// Disclaimer
// 
// This publication contains statements about the suitability of our products for certain areas of application. These statements are based on typical features of our products. The examples shown in this publication are for demonstration purposes only. 
// The information provided herein should not be regarded as specific operation characteristics. It is incumbent on the customer to check and decide whether a product is suitable for use in a particular application. 
// We do not give any warranty that the source code which is made available with this publication is complete or accurate. 
//
// THE SAMPLE CODE CONTAINED IN THIS PUBLICATION IS PROVIDED “AS IS” WITHOUT WARRANTY OF ANY KIND, EITHER EXPRESSED, IMPLIED OR STATUTORY, INCLUDING WITHOUT LIMITATION, ANY WARRANTY WITH RESPECT TO NON-INFRINGEMENT, FREEDOM FROM PROPRIETARY RIGHTS OF THIRD PARTIES OR FITNESS FOR ANY PARTICULAR PURPOSE. 
// This publication may be changed from time to time without prior notice. No liability is assumed for errors and/or omissions. Our products are described in detail in our data sheets and documentations. Product-specific warnings and cautions must be observed. 
// For the latest version of our data sheets and documentations visit our website (www.beckhoff.de). 
//
// © Beckhoff Automation GmbH & Co. KG, 2022
// The reproduction, distribution and utilization of this document as well as the communication of its contents to others without express authorization is prohibited. Offenders will be held liable for the payment of damages. All rights reserved in the event of the grant of a patent, utility model or design.
PROGRAM MAIN
VAR_INPUT
	bExecuteComplete			: BOOL;									//Command Execute Complete, not defined
END_VAR
VAR
	UserModeCofig				: PML_UnitModeConfig;					//User can configure his own Mode
	
	fbMachine					: FB_Machine;							//Instance of FB_Machine
	bMachineStartedUp			: BOOL := FALSE;						//TRUE, when first PLC-Cycle finish

	fbVisu						: FB_Visu;								//Visualization
	
	fbTrigger					: F_TRIG;								//Trigger for resseting Counters

	fbLocalSystemTime			 : FB_LocalSystemTime;					//Get local Systemtime
	
	fbTriggerErrorMainAxis		: R_TRIG;								//Trigger for detecting Error on Mainaxis and write into PackTags
	fbTriggerErrorMetalAxis		: R_TRIG;								//Trigger for detecting Error on Metalaxis and write into PackTags
	fbTriggerErrorPlasticAxis	: R_TRIG;								//Trigger for detecting Error on Plasticaxis and write into PackTags
	
	nStateCommandCheck			: DINT;									//State to handle with statecommands
	
	i	: INT;
	tonDly	: TON;
	
	fb_ups	:FB_S_UPS_CX51x0;
	application	: FB_Application;

	bButton				: BOOL;
	ton_button			: TON;

	refMachine_control_cmd	:REFERENCE TO MachineControlCommand;
	
	
	PackTags					: ST_PackMLv30;	
	rTrig_error	:ARRAY[0..10] OF R_TRIG;
	rTrig_agingTest	:R_TRIG;
	fTrig_agingTest	:F_TRIG;
	refStates_fb_roller_0 : REFERENCE TO E_RollerStates;
	refStates_fb_roller_1 : REFERENCE TO E_RollerStates;
	refStates_fb_roller_2 : REFERENCE TO E_RollerStates;
	refStates_fb_roller_3 : REFERENCE TO E_RollerStates;
	refStates_fb_loading  : REFERENCE TO E_LoadingStates;
	refStates_fb_working  : REFERENCE TO E_WorkingStates;
	
	
	
END_VAR

fb_ups();
GVL.fb_mcp();

application();
refMachine_control_cmd	REF= MAIN.application.tote_subsystem.machine_control_cmd;

tonDly(PT:= T#10MS);
//Configure Usermode 1
A_UnitModeConfig();

//Runs the first PLC-Cycle
IF fbMachine.bUndefinedDone AND NOT bMachineStartedUp THEN
	GVL.PackTags.Command.CntrlCmd	:= ePMLCommand_Abort;
	bMachineStartedUp			:= TRUE;
END_IF


GVL.bButtonProductionReq := GVL.PackTags.Command.UnitMode = ePMLProtUnitMode_Production AND GVL.PackTags.Status.UnitModeCurrent <> GVL.PackTags.Command.UnitMode;


CASE nStateCommandCheck OF	
0:
	tonDly.IN := FALSE;
	GVL.PackTags.Command.CntrlCmd := ePMLCommand_Undefined;
	nStateCommandCheck :=1;
1:	
	tonDly.IN := TRUE;
	IF tonDly.Q THEN
		nStateCommandCheck :=0;
	END_IF
CASE fbMachine.eState OF
			
	ePMLState_Aborted:
		IF (GVL.PackTags.Command.CntrlCmd = ePMLCommand_Clear OR GVL.fb_mcp.st_safety_door.button_reset) THEN
			fbMachine.eCommand	:= ePMLCommand_Clear;
		END_IF
	ePMLState_Complete:		
		IF (GVL.PackTags.Command.CntrlCmd = ePMLCommand_Reset OR refMachine_control_cmd = MachineControlCommand.RESET OR GVL.fb_mcp.st_safety_door.button_reset) THEN
			fbMachine.eCommand	:= ePMLCommand_Reset;
		END_IF
	ePMLState_Idle:
		IF (GVL.PackTags.Command.CntrlCmd = ePMLCommand_Start OR refMachine_control_cmd = MachineControlCommand.START)	
	 	AND (NOT (GVL.PackTags.Command.Parameter[1].Value <= 0) OR NOT (fbMachine.eMode = 1))THEN
			 fbMachine.eCommand	:= ePMLCommand_Start; 
		END_IF
		IF refMachine_control_cmd = MachineControlCommand.RESET THEN
			refMachine_control_cmd	:= MachineControlCommand.DO_NOTHING;
		END_IF
	ePMLState_Stopped:
		IF (GVL.PackTags.Command.CntrlCmd = ePMLCommand_Reset OR refMachine_control_cmd = MachineControlCommand.RESET OR GVL.fb_mcp.st_safety_door.button_reset) THEN
			fbMachine.eCommand	:= ePMLCommand_Reset;
		END_IF		
		IF (GVL.PackTags.Command.CntrlCmd = ePMLCommand_Start OR refMachine_control_cmd = MachineControlCommand.START)	
	 	AND (NOT (GVL.PackTags.Command.Parameter[1].Value <= 0) OR NOT (fbMachine.eMode = 1))
		AND stPMLUnitModeConfiguration[fbMachine.eMode].aStateDisabled[ePMLState_Idle] THEN
			fbMachine.eCommand	:= ePMLCommand_Start; 
		END_IF	
		IF refMachine_control_cmd = MachineControlCommand.STOP THEN
			refMachine_control_cmd	:= MachineControlCommand.DO_NOTHING;
		END_IF	
	ePMLState_Execute:	
		IF refMachine_control_cmd = MachineControlCommand.START THEN
			refMachine_control_cmd	:= MachineControlCommand.DO_NOTHING;
		END_IF
		IF GVL.PackTags.Command.CntrlCmd = ePMLCommand_Hold		
		AND( fbMachine.eMode =  1 OR fbMachine.eMode =  4 OR fbMachine.eMode = 2)  THEN
			fbMachine.eCommand	:= ePMLCommand_Hold;
		END_IF	
		IF GVL.PackTags.Command.CntrlCmd = ePMLCommand_Suspend	
		AND (fbMachine.eMode = 4 OR fbMachine.eMode = 1)THEN
			fbMachine.eCommand	:= ePMLCommand_Suspend;
		END_IF	 
	ePMLState_Held:	 
		IF GVL.PackTags.Command.CntrlCmd = ePMLCommand_Unhold THEN
			fbMachine.eCommand	:= ePMLCommand_Unhold;
		END_IF
	ePMLState_Suspended:
		IF GVL.PackTags.Command.CntrlCmd = ePMLCommand_Unsuspend THEN
		 	fbMachine.eCommand	:= ePMLCommand_Unsuspend;
		END_IF
	
END_CASE

/////////////////////////////abort/////////////////////////////	
IF 	fbMachine.eState <> ePMLState_Aborted AND fbMachine.eState <> ePMLState_Clearing THEN	
	IF GVL.PackTags.Command.CntrlCmd = ePMLCommand_Abort OR M_CheckError() THEN
		fbMachine.eCommand	:= ePMLCommand_Abort;
		refMachine_control_cmd	:= MachineControlCommand.DO_NOTHING;
	END_IF
END_IF
/////////////////////////////stop/////////////////////////////					
IF (GVL.PackTags.Command.CntrlCmd = ePMLCommand_Stop OR refMachine_control_cmd = MachineControlCommand.STOP) THEN
	fbMachine.eCommand	:= ePMLCommand_Stop;
	//
END_IF


2:
;
END_CASE



//
//Set the Packtags
M_SetPackTags();

//set the errors and warnings in Packtags
M_SetPackTagsErrorWarning();

//Call Visu
M_CallVisu();
///////////////////initialize unitmode and set 
IF GVL.PackTags.Command.UnitMode=ePMLProtUnitMode_Invalid THEN
	GVL.PackTags.Command.UnitMode	:= ePMLProtUnitMode_Production;
	GVL.PackTags.Command.Parameter[1].Value := 1;
END_IF
//Call FB_Machine
fbMachine(eModeCommand:= GVL.PackTags.Command.UnitMode,  eMode => GVL.PackTags.Status.UnitModeCurrent, eState =>GVL.PackTags.Status.StateCurrent);

ACTION A_UnitModeConfig:
UserModeCofig(
	eMode							:= ePMLUnitMode_Service, 
	bDisableClearing				:= TRUE, 
	bDisableStarting				:= FALSE, 
	bDisableSuspended				:= FALSE, 
	bDisableStopping				:= TRUE, 
	bDisableAborting				:= TRUE, 
	bDisableHolding					:= TRUE, 
	bDisableHeld					:= TRUE, 
	bDisableUnholding				:= TRUE, 
	bDisableSuspending				:= TRUE, 
	bDisableUnsuspending			:= TRUE, 
	bDisableResetting				:= TRUE, 
	bDisableIdle					:= FALSE, 
	bDisableCompleting				:= TRUE, 
	bDisableComplete				:= FALSE, 
	bEnableUnitModeChangeStopped	:= TRUE, 
	bEnableUnitModeChangeIdle		:= TRUE, 
	bEnableUnitModeChangeSuspended	:= FALSE, 
	bEnableUnitModeChangeExecute	:= FALSE, 
	bEnableUnitModeChangeAborted	:= TRUE, 
	bEnableUnitModeChangeHeld		:= FALSE, 
	bEnableUnitModeChangeComplete	:= TRUE, 
	bError							=> , 
	nErrorId						=> );
END_ACTION

METHOD M_CallVisu
VAR_INPUT
END_VAR
//Calling FB_Visu
fbVisu(

	aKeyPressed				:= GVL.aKeyPressed,
	aUnitInfo				:= GVL.aUnitInfo, 
	bInvalidEntry			=> ,
	aCaption				=> GVL.aCaption,
	eModeVisu				=> ,
	eStateVisu				=> ,
	sUnitName				=> ,
	iFrameVisible			=> );
END_METHOD

METHOD M_CheckError : BOOL
VAR_INPUT
END_VAR

VAR
	
	
END_VAR
M_CheckError	:= FALSE;
FOR i:=1 TO GlobalParameters.MaxAlarms DO
	IF GVL.PackTags.Admin.Alarm[i].Trigger THEN
		M_CheckError	:= TRUE;
	END_IF
END_FOR
RETURN;//remove this while safety and air is ready
rTrig_error[0]();
rTrig_error[1]();
IF GVL.PackTags.Status.StateCurrent<>E_PMLState.ePMLState_Resetting THEN
	FOR i:=0 TO 10 DO
		IF rTrig_error[i].Q THEN
			GVL.pml_adminAlarm.M_SetAlarm(stAdmin:=GVL.PackTags.Admin,stAlarm:=GVL.alarm);
		END_IF
	END_FOR
END_IF

IF application.air_pressure_subsystem.current_air_pressure_state=CurrentAirPressureState.ERROR THEN
	GVL.alarm.Message	:= 'Air pressure is low';
	rTrig_error[0].CLK	:= TRUE;
ELSE
	rTrig_error[0].CLK	:= FALSE;
END_IF
IF application.safety.xError THEN
	GVL.alarm.Message	:= 'Safety input trigger';
	rTrig_error[1].CLK	:= TRUE;
ELSE
	rTrig_error[1].CLK	:= FALSE;
END_IF


IF application.safety.xError OR application.air_pressure_subsystem.current_air_pressure_state=CurrentAirPressureState.ERROR THEN
	M_CheckError	:= TRUE;
END_IF
END_METHOD

METHOD M_SetPackTags
VAR_INPUT
END_VAR
VAR	
END_VAR
//***************************Writing Data into GVL.PackTags***************************

//Parameters for the production
GVL.PackTags.Command.Parameter[1].ID				:= 1;
GVL.PackTags.Command.Parameter[1].Name				:= 'Quantity';
GVL.PackTags.Command.Parameter[1].Unit				:= 'Tote';

//Countig produced totes, see FB_sample
GVL.PackTags.Admin.ProdProcessedCount[1].ID			:= 1;
GVL.PackTags.Admin.ProdProcessedCount[1].Name		:= 'ToteFinish_Sample';
GVL.PackTags.Admin.ProdProcessedCount[1].Unit		:= 'Tote';





//Write the actual state and mode into the GVL.PackTags
GVL.PackTags.Status.StateCurrent					:= fbMachine.eState;
GVL.PackTags.Status.UnitModeCurrent					:= fbMachine.eMode;
GVL.PackTags.Status.StateRequested					:= fbMachine.eCommand;
GVL.PackTags.Status.UnitModeRequested				:= fbMachine.eModeCommand;
GVL.PackTags.Status.StateChangeInProcess			:= GVL.PackTags.Status.StateCurrent <> GVL.PackTags.Status.StateRequested;
GVL.PackTags.Status.UnitModeChangeInProcess			:= GVL.PackTags.Status.UnitModeCurrent <> GVL.PackTags.Status.UnitModeRequested;

//Write actual time and date in GVL.PackTags
fbLocalSystemTime(sNetID:= '', bEnable := TRUE);
GVL.PackTags.Admin.PlcDateTime[0]	:= fbLocalSystemTime.systemTime.wYear;
GVL.PackTags.Admin.PlcDateTime[1]	:= fbLocalSystemTime.systemTime.wMonth;
GVL.PackTags.Admin.PlcDateTime[2]	:= fbLocalSystemTime.systemTime.wDay;
GVL.PackTags.Admin.PlcDateTime[3]	:= fbLocalSystemTime.systemTime.wHour;
GVL.PackTags.Admin.PlcDateTime[4]	:= fbLocalSystemTime.systemTime.wMinute;
GVL.PackTags.Admin.PlcDateTime[5]	:= fbLocalSystemTime.systemTime.wSecond;
GVL.PackTags.Admin.PlcDateTime[6]	:= fbLocalSystemTime.systemTime.wMilliseconds;


//Set the productcounter to 0, when the production command is completed
fbTrigger(CLK:= (fbMachine.eState = ePMLState_Complete));
IF fbTrigger.Q OR GVL.stChangeIntoProduction.bYesReset THEN
	GVL.PackTags.Admin.ProdProcessedCount[1].Count	:= 0;
	GVL.PackTags.Command.Parameter[1].Value			:= 0;
	GVL.nVisuProductCommand							:= 0;
END_IF
END_METHOD

METHOD M_SetPackTagsErrorWarning
VAR_INPUT
END_VAR
//====================Error and Warnig setting========================
//Warnings
GVL.PackTags.Admin.Warning[1].Message	:= 'Invalid Production Command, command Products must be higher than 0';
GVL.PackTags.Admin.Warning[1].ID 		:= 1;

GVL.PackTags.Admin.Warning[2].Message	:= 'Invalid Mode Command, please try anothereone';
GVL.PackTags.Admin.Warning[2].ID		:= 2;


//====================Error and Warnig handling========================
//warning for invalid production command
IF GVL.PackTags.Status.UnitModeCurrent = ePMLProtUnitMode_Production AND GVL.PackTags.Status.StateCurrent = ePMLState_Idle AND GVL.PackTags.Command.CntrlCmd = ePMLCommand_Start AND GVL.PackTags.Command.Parameter[1].Value <= 0 THEN
	GVL.PackTags.Admin.Warning[1].Trigger :=TRUE;
ELSE
	GVL.PackTags.Admin.Warning[1].Trigger :=FALSE;
END_IF

//warning for invalid mode command
IF fbMachine.bInvalidModeCommandOut THEN
	GVL.PackTags.Admin.Warning[2].Trigger :=TRUE;
ELSE 
	GVL.PackTags.Admin.Warning[2].Trigger :=FALSE;
END_IF
END_METHOD

END_PROGRAM

(* stored: Version 1.1.0.1, ProductVersion 3.1.4024.12
   POU MAIN: Id {3db2f275-2958-4d55-b639-7561aac45e5f}, SpecialFunc None
   Action A_UnitModeConfig: Id {22b649e9-a085-4601-8ad9-54522ade47b0}
   Method M_CallVisu: Id {1e59b2a3-52d5-45b9-816e-b9175fe8bcf5}
   Method M_CheckError: Id {d8e49d3a-3d8f-42dd-85ad-c6bb140b7f9b}
   Method M_SetPackTags: Id {e3fcccbd-b9f1-4f18-9b86-975dcfc89c23}
   Method M_SetPackTagsErrorWarning: Id {9cf9563e-0860-4b80-8190-1adefae96c7f} *)
